FUNCTION_BLOCK Organization_Services (* Basic Function Block Type *)
  (* Standard: 61499-2 *)
  (* Version 0.0, 11/2/2020, prana, nxtControl GmbH, Template *)
  PACKAGE Main;
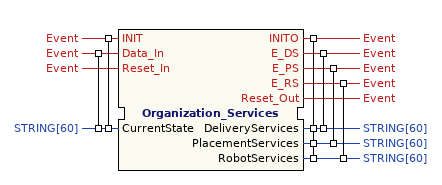
  EVENT_INPUT
    INIT WITH CurrentState; (* Initialization Request *)
    Data_In WITH CurrentState;
    Reset_In;
  END_EVENT
  EVENT_OUTPUT
    INITO WITH DeliveryServices, PlacementServices, RobotServices; (* Initialization Confirm *)
    E_DS WITH DeliveryServices;
    E_PS WITH PlacementServices;
    E_RS WITH RobotServices;
    Reset_Out;
  END_EVENT
  VAR_INPUT
    CurrentState : STRING[60];
  END_VAR
  VAR_OUTPUT
    DeliveryServices : STRING[60];
    PlacementServices : STRING[60];
    RobotServices : STRING[60];
  END_VAR
  VAR
    DS : BOOL;
    PS : BOOL;
    check : STRING[60];
    RS : BOOL;
  END_VAR
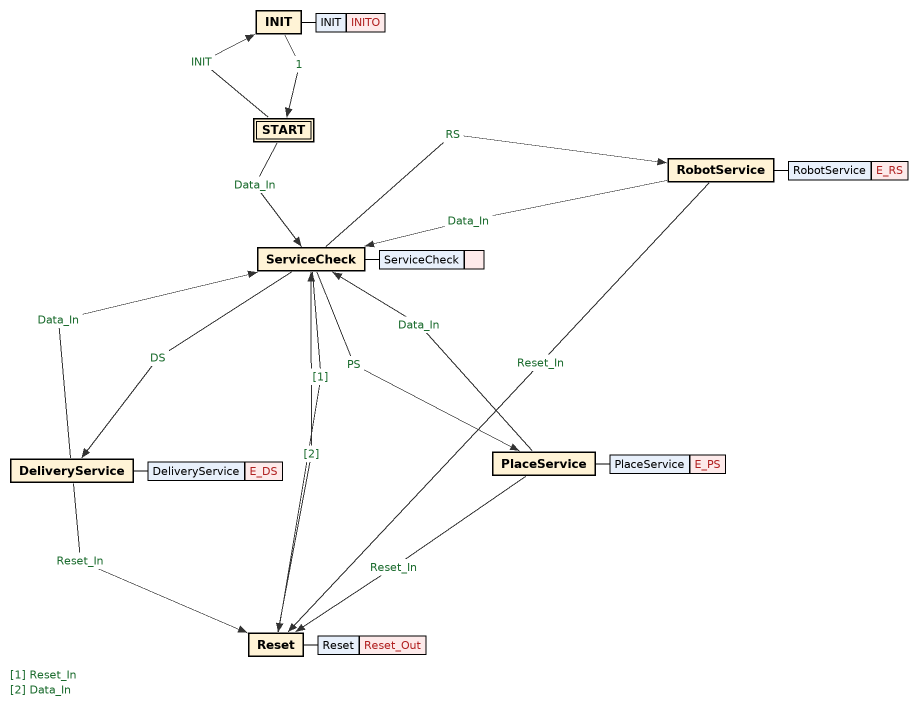
  EC_STATES
    START; (* Initial State *)
    INIT : INIT -> INITO; (* Initialization *)
    ServiceCheck : ServiceCheck;
    DeliveryService : DeliveryService -> E_DS;
    PlaceService : PlaceService -> E_PS;
    Reset : Reset -> Reset_Out;
    RobotService : RobotService -> E_RS;
  END_STATES
  EC_TRANSITIONS
    START TO INIT := INIT;
    INIT TO START := 1;
    START TO ServiceCheck := Data_In;
    ServiceCheck TO DeliveryService := DS;
    ServiceCheck TO PlaceService := PS;
    DeliveryService TO ServiceCheck := Data_In;
    PlaceService TO ServiceCheck := Data_In;
    PlaceService TO Reset := Reset_In;
    DeliveryService TO Reset := Reset_In;
    Reset TO ServiceCheck := Data_In;
    ServiceCheck TO Reset := Reset_In;
    ServiceCheck TO RobotService := RS;
    RobotService TO ServiceCheck := Data_In;
    RobotService TO Reset := Reset_In;
  END_TRANSITIONS
  ALGORITHM INIT IN ST: (* Initialization algorithm *)
;
  END_ALGORITHM
  ALGORITHM Reset IN ST: (* Normally executed algorithm *)
check := '';

DS := FALSE;
PS := FALSE;
RS := FALSE;
  END_ALGORITHM
  ALGORITHM ServiceCheck IN ST:
check := (LEFT(CurrentState,1));
IF check = 'C' THEN
	DS := TRUE;
    PS := FALSE;
    RS := FALSE;
ELSIF check = 'J' THEN
	PS := TRUE;
	DS := FALSE;
	RS := FALSE;
ELSIF check = 'R' THEN
	RS := TRUE;
	DS := FALSE;
	PS := FALSE;
END_IF;
  END_ALGORITHM
  ALGORITHM DeliveryService IN ST:
DeliveryServices := CurrentState;
DS := FALSE;
PS := FALSE;
RS := FALSE;
Data_In := FALSE;
PlacementServices := '';
  END_ALGORITHM
  ALGORITHM PlaceService IN ST:
PlacementServices := CurrentState;
DS := FALSE;
PS := FALSE;
RS := FALSE;
Data_In := FALSE;
DeliveryServices := '';
  END_ALGORITHM
  ALGORITHM RobotService IN ST:
RobotServices := CurrentState;

DS := FALSE;
PS := FALSE;
RS := FALSE;
Data_In := FALSE;
DeliveryServices := '';
  END_ALGORITHM
END_FUNCTION_BLOCK
